// TIA Portal project "3rd_Party_Server" (V14)

(* hardware
DEVICE "S7-1200 station_1"  S7-1200 Station
   slot 0: "Rack_0"  S7-1200 Rack  Rack  V1.0
   slot 1: "PLC_1"  CPU 1212C DC/DC/DC  6ES7 212-1AE40-0XB0  V4.2
*)

// ===== PLC "PLC_1"  CPU 1212C DC/DC/DC =====

DATA_BLOCK "3rd_Party_Data"   // DB101
{ S7_Optimized_Access := 'FALSE' }
VERSION : 0.1
   VAR
      主控_通讯检查 : Array[0..7] of Bool;
      主控_备用_BYTE_2 : Byte;
      主控_备用_BYTE_3 : Byte;
      主控_备用_BYTE_4 : Byte;
      主控_系统急停_急停 : Bool;   // 急停，上升沿触发
      主控_系统急停_急停复位 : Bool;   // 急停复位
      主控_系统急停_备用_1 : Bool;
      主控_系统急停_备用_2 : Bool;
      主控_系统急停_备用_3 : Bool;
      主控_系统急停_备用_4 : Bool;
      主控_系统急停_备用_5 : Bool;
      主控_系统急停_备用_6 : Bool;
      主控_备用_Word_6 : Word;
      主控_备用_Word_8 : Word;
      主控_任务_种类编码 : Word;   // 2^15种
      主控_任务_任务状态 : Word;   // 同上次比较
      主控_任务_起点信息 : Word;   // 取料工位
      主控_任务_终点信息 : Word;   // 放料工位
      主控_任务_其他任务信息 : Word;
      主控_备用_Word_20 : Word;
      主控_备用_Word_22 : Word;
      主控_备用_Word_24 : Word;
      主控_备用_Word_26 : Word;
      主控_备用_Word_28 : Word;
      主控_To_AGV_Signal : Array[0..200] of Bool;
      主控_备用_Word_56 : Word;
      主控_From_AGV_Signal_1 : Array[0..310] of Bool;
      主控_备用_Word_98 : Word;
      主控_扩展信号 : Array[0..49] of Word;
      过渡空信号 : Array[0..49] of Word;
      AGV_PLC通信 : Array[0..15] of Bool;
      AGV_备用_Word_302_308 : Array[0..3] of Word;
      AGV_任务接收确认 : Word;   // 任务收到信号
      AGV_任务确认信息1 : Word;
      AGV_任务确认信息2 : Word;   // 高字节： AGV# ； 低字节： error bit标识： 【0：通讯故障； 1： CAN网络故障；2： 碰撞触发； 3：急停 ； 4：伺服故障； 5：脱磁故障 ；6：插齿未插到料 ； 】
      AGV_备用_Word_316 : Word;
      AGV_备用_Word_318 : Word;
      AGV_OuterSignal确认 : Array[1..200] of Word;
      AGV_扩展确认信号 : Array[1..50] of Word;
      AGV_备用_Word_720 : Array[1..15] of Word;
      AGV_AGV错误上报 : Array[1..10] of Word;
      "AGV_请求上报信号(Word)" : Array[1..100] of Word;
      "AGV_请求上报信号(DWord)" : Array[101..300] of DWord;
      AGV_备用_Word_1350 : Array[0..29] of Word;
   END_VAR
BEGIN
   // 主控_通讯检查[0] : 心跳，1s周期
   // 主控_通讯检查[1] : 备用
   // 主控_通讯检查[2] : 备用
   // 主控_通讯检查[3] : 备用
   // 主控_通讯检查[4] : 备用
   // 主控_通讯检查[5] : 备用
   // 主控_通讯检查[6] : 备用
   // 主控_通讯检查[7] : 备用
   // 主控_To_AGV_Signal[0] : 1#呼叫换货架
   // 主控_To_AGV_Signal[1] : 2#呼叫换货架
   // 主控_To_AGV_Signal[2] : 卷帘门开到位
   // 主控_To_AGV_Signal[3] : 卷帘门关到位
   // 主控_To_AGV_Signal[4] : 1#允许顶升
   // 主控_To_AGV_Signal[5] : 2#允许顶升
   // 主控_From_AGV_Signal_1[0] : 错误上报信号1
   // 主控_From_AGV_Signal_1[1] : 错误上报信号2
   // 主控_From_AGV_Signal_1[2] : 错误上报信号3
   // 主控_From_AGV_Signal_1[3] : 错误上报信号4
   // 主控_From_AGV_Signal_1[4] : 错误上报信号5
   // 主控_From_AGV_Signal_1[5] : 错误上报信号6
   // 主控_From_AGV_Signal_1[6] : 错误上报信号7
   // 主控_From_AGV_Signal_1[7] : 错误上报信号8
   // 主控_From_AGV_Signal_1[8] : 错误上报信号9
   // AGV_PLC通信[0] : 1s脉冲心跳信号
   // AGV_PLC通信[1] : 备用
   // AGV_PLC通信[2] : 备用
   // AGV_PLC通信[3] : 备用
   // AGV_PLC通信[4] : 备用
   // AGV_PLC通信[5] : 备用
   // AGV_PLC通信[6] : 备用
   // AGV_PLC通信[7] : 备用
   // AGV_PLC通信[8] : 备用
   // "AGV_请求上报信号(Word)"[1] : 1#货架更换完成
   // "AGV_请求上报信号(Word)"[2] : 2#货架更换完成
   // "AGV_请求上报信号(Word)"[3] : 请求开卷帘门
   // "AGV_请求上报信号(Word)"[4] : 请求关卷帘门
   // "AGV_请求上报信号(Word)"[5] : 7#-10#满料信号
   // "AGV_请求上报信号(Word)"[6] : 1#报警
   // "AGV_请求上报信号(Word)"[7] : 2#报警
   // "AGV_请求上报信号(DWord)"[101] : 示例：工位到达 （第一个字： AGV#， 第二个字： Point#）
   // "AGV_请求上报信号(DWord)"[102] : 示例：（第一个字： AGV#空闲； 第二个字： 处于位置point#）
END_DATA_BLOCK

ORGANIZATION_BLOCK "Main"   // OB1, LAD, ProgramCycle
TITLE = "Main Program Sweep (Cycle)"
{ S7_Optimized_Access := 'TRUE' }
VERSION : 0.1
   VAR_INPUT
      Initial_Call : Bool;   // Initial call of this OB
      Remanence : Bool;   // =True, if remanent data are available
   END_VAR
BEGIN
END_ORGANIZATION_BLOCK